// Core §2.2 — discrete-command composite tier. Child recursion lives in
// FB_CompositeModuleBase; this type supplies Equipment Module identity/capability.
FUNCTION_BLOCK ABSTRACT FB_EquipmentModuleBase EXTENDS FB_CompositeModuleBase IMPLEMENTS I_EquipmentModule

PROPERTY ModuleType : E_ModuleType
GET
ModuleType := E_ModuleType.EQUIPMENT_MODULE;
END_GET
END_PROPERTY

END_FUNCTION_BLOCK

(* stored: Version 1.1.0.1, ProductVersion 3.1.4024.12
   POU FB_EquipmentModuleBase: Id {90f86e09-a7f8-40f2-ad09-f70330a42249}, SpecialFunc None
   Property ModuleType: Id {381e8308-5bcb-40ca-9818-8a883dc4cf03}
   Get Get: Id {e46489ac-bd20-4bac-b0ef-28c89566d47d} *)
